TYPE E_MachineState :
STRUCT

END_STRUCT
END_TYPE

(* stored: Version 1.1.0.1, ProductVersion 3.1.4024.16
   DUT E_MachineState: Id {d11e1d8f-51f0-4036-9189-8bde2e0915ed} *)
